FUNCTION_BLOCK ADD_SINT (* IEC 61131-3 SINT Addition *)
  (* Standard: 61131-3 *)
  (* Version 0.0, 2004-12-15, JHC, Rockwell Automation, Converted from SRC format. *)
  (* Compiler header: package fb.rt.plc.math; *)
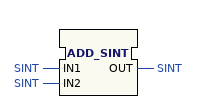
  VAR_INPUT
    IN1 : SINT; (* Augend *)
    IN2 : SINT; (* Addend *)
  END_VAR
  VAR_OUTPUT
    OUT : SINT; (* Sum *)
  END_VAR
END_FUNCTION_BLOCK
